(* IEC 61131-3 sources: POMIRTS_lab3/AS/Library_2/AsFifo, 3 files *)

(* ---- AsFifo.typ ---- *)
TYPE

END_TYPE

(* ---- AsFifo.fun ---- *)
{REDUND_CONTEXT} {REDUND_UNREPLICABLE} FUNCTION_BLOCK fifoCreate (*creates a fifo; asynchronous execution*)
	VAR_INPUT
		enable : BOOL; (*enables execution*)
		pFifo : UDINT; (*fifo name given as a pointer. Max. 32 charachter are allowed*)
		size : UDINT; (*size of the fifo in bytes*)
		mode : UINT; (*write mode (fifoMODE_WRITE_UNTIL_FULL,  fifoMODE_WRITE_UNTIL_FULL)*)
	END_VAR
	VAR_OUTPUT
		status : UINT; (*execution status: ERR_OK, ERR_FUB_ENABLE_FALSE, ERR_FUB_BUSY, 0xXXXX = see help*)
		ident : UDINT; (*identifier of the fifo*)
	END_VAR
	VAR
		i_state : UINT; (*internal variable*)
		i_result : UINT; (*internal variable*)
		i_tmp : UDINT; (*internal variable*)
	END_VAR
END_FUNCTION_BLOCK

{REDUND_CONTEXT} {REDUND_UNREPLICABLE} FUNCTION_BLOCK fifoDelete (*deletes a  fifo; asynchronous execution*)
	VAR_INPUT
		enable : BOOL; (*enables execution*)
		ident : UDINT; (*fifo ident*)
	END_VAR
	VAR_OUTPUT
		status : UINT; (*execution status: ERR_OK, ERR_FUB_ENABLE_FALSE, ERR_FUB_BUSY, 0xXXXX = see help*)
	END_VAR
	VAR
		i_state : UINT; (*internal variable*)
		i_result : UINT; (*internal variable*)
		i_tmp : UDINT; (*internal variable*)
	END_VAR
END_FUNCTION_BLOCK

{REDUND_CONTEXT} {REDUND_UNREPLICABLE} FUNCTION_BLOCK fifoWrite (*writes data into fifo; synchronous execution*)
	VAR_INPUT
		enable : BOOL; (*enables execution*)
		ident : UDINT; (*fifo ident*)
		pData : UDINT; (*fifo data source given as a pointer*)
		size : UDINT; (*size of fifo data in bytes*)
	END_VAR
	VAR_OUTPUT
		status : UINT; (*execution status: ERR_OK, ERR_FUB_ENABLE_FALSE 0xXXXX = see help*)
	END_VAR
	VAR
		i_tmp : UDINT; (*internal variable*)
	END_VAR
END_FUNCTION_BLOCK

{REDUND_CONTEXT} {REDUND_UNREPLICABLE} FUNCTION_BLOCK fifoRead (*reads data from fifo; synchronous execution*)
	VAR_INPUT
		enable : BOOL; (*enables execution*)
		ident : UDINT; (*fifo ident*)
		pData : UDINT; (*fifo data source given as a pointer*)
		size : UDINT; (*size of fifo data in bytes*)
	END_VAR
	VAR_OUTPUT
		status : UINT; (*execution status: ERR_OK, ERR_FUB_ENABLE_FALSE  0xXXXX = see help*)
	END_VAR
END_FUNCTION_BLOCK

{REDUND_CONTEXT} {REDUND_UNREPLICABLE} FUNCTION_BLOCK fifoClear (*clears all data of fifo; asynchronous execution*)
	VAR_INPUT
		enable : BOOL; (*enables execution*)
		ident : UDINT; (*fifo ident*)
	END_VAR
	VAR_OUTPUT
		status : UINT; (*execution status: ERR_OK, ERR_FUB_ENABLE_FALSE, ERR_FUB_BUSY, 0xXXXX = see help*)
	END_VAR
	VAR
		i_state : UINT; (*internal variable*)
		i_result : UINT; (*internal variable*)
		i_tmp : UDINT; (*internal variable*)
	END_VAR
END_FUNCTION_BLOCK

{REDUND_CONTEXT} {REDUND_UNREPLICABLE} FUNCTION_BLOCK fifoGetInfo (*gets fifo info; synchronous execution*)
	VAR_INPUT
		enable : BOOL; (*enables execution*)
		ident : UDINT; (*fifo ident*)
	END_VAR
	VAR_OUTPUT
		status : UINT; (*execution status: ERR_OK, ERR_FUB_ENABLE_FALSE, 0xXXXX = see help*)
		fifoFree : UDINT; (*value of free bytes*)
		fifoUsed : UDINT; (*value of used bytes*)
	END_VAR
END_FUNCTION_BLOCK

{REDUND_CONTEXT} {REDUND_UNREPLICABLE} FUNCTION fifoGetIdent : UDINT (*status: ERR_OK,  0xXXXX = see help*)
	VAR_INPUT
		pFifo : UDINT; (*fifo name given as a pointer*)
		pIdent : UDINT; (*fifo ident*)
	END_VAR
END_FUNCTION

(* ---- AsFifo.var ---- *)
VAR CONSTANT
	fifoERR_INVALID_PARAM : UINT := 36780; (*check parameters. At least one of needed ones is zero*)
	fifoERR_INVALID_IDENT : UINT := 36781; (*invalid fifo ident, check parameters*)
	fifoERR_INVALID_MODE : UINT := 36782; (*error mode*)
	fifoERR_FIFO_ALREADY_EXISTS : UINT := 36783; (*fifo with this name already exists*)
	fifoERR_FIFO_NOT_EXIST : UINT := 36784; (*fifo not exist*)
	fifoERR_FIFO_LIST_FULL : UINT := 36785; (*maximal amount of fifo reached*)
	fifoERR_BUFFER_FULL : UINT := 36786; (*buffer is full error*)
	fifoERR_BUFFER_EMPTY : UINT := 36787; (*buffer is empty*)
	fifoERR_SYSTEM : UINT := 36788; (*internal error*)
	fifoMODE_WRITE_UNTIL_FULL : UINT := 1; (*writes only until fifo is full, no overwrite*)
	fifoMODE_WRITE_ALWAYS : UINT := 2; (*writes always, overwrites*)
END_VAR
